TYPE EL3078_EX EXTENDS EL3078 :
STRUCT
	WcState AT %I* : BOOL;
	InputToggle AT %I* : BOOL;
	State AT %I* : UINT;
	AdsAdr AT %I* : Global.AMSADDR;
END_STRUCT
END_TYPE

(* stored: Version 1.1.0.1, ProductVersion 3.1.4026.18
   DUT EL3078_EX: Id {0f135d0e-d858-4371-8e5e-53474f4a5138} *)
